FUNCTION_BLOCK Stagger_FB

VAR_INPUT
	start : BOOL := FALSE;
	n	  : INT := 8;
	reset : BOOL := FALSE;
END_VAR
VAR
	delayTMR_TON : TON;
	delayTMR_PT	 : TIME := T#100MS;
	delayTMR_ET	 : TIME;
	state		 : INT := 0;
	i			 : INT := 1;
	
	startOutput  : BOOL := 0;
END_VAR
VAR_OUTPUT
	OutputHi	: ARRAY[1..8] OF BOOL;

END_VAR

(* start goes high, stagger output sequence starts in a delay, 
	when the last output is high, it goes to idle,
	if reset goes high, it turns off all outputs - this fb needs to be reset when we dont want to output to be high.
	**to add, if both start and reset are high, throw a warning sign
*)
IF start = TRUE THEN 

CASE state OF
	0: 	//idle 	
//		FOR i := 1 TO n BY 1 DO 
//			OutputHi[i] := FALSE;
//		END_FOR
		delayTMR_TON (IN := FALSE, PT := delayTMR_PT, ET => delayTMR_ET);
		IF start = TRUE THEN 
			state := 1;
//			ELSIF reset = TRUE THEN 
//				state := 3;
//			ELSE 
//				state := 0;
		END_IF
		
	1: 	//output
		OutputHi[i] := TRUE;
		delayTMR_TON (IN := TRUE, PT := delayTMR_PT, ET => delayTMR_ET);
		
		IF delayTMR_TON.Q = TRUE THEN 
			state := 2;
		END_IF;
	2:	//increment
		delayTMR_TON (IN := FALSE, PT := delayTMR_PT, ET => delayTMR_ET);
		i := i + 1;
		
		IF OutputHi[n] = TRUE THEN 
			start := FALSE;
			state := 0;
		ELSE 
			IF i > n THEN 
				i := 1;
			END_IF
			state := 1;
		END_IF;
//	3:	//reset output 
//		FOR i := 1 TO n BY 1 DO 
//			OutputHi[i] := FALSE;
//		END_FOR
//		delayTMR_TON (IN := FALSE, PT := delayTMR_PT, ET => delayTMR_ET);
//		reset := 0; //debounce reset input
//		state := 0;
END_CASE

ELSIF reset = TRUE THEN 
		FOR i := 1 TO n BY 1 DO 
			OutputHi[i] := FALSE;
		END_FOR
		i := 1;
		state := 0;
END_IF;

IF i > n THEN 
	i := 1;
END_IF

END_FUNCTION_BLOCK

(* stored: Version 1.1.0.1, ProductVersion 3.1.4024.11
   POU Stagger_FB: Id {f66eca1b-eacb-46d0-ae51-b07877c95021}, SpecialFunc None *)
